SUBAPPLICATION Uebung_237_AX (* AD_TO_AR-Bitfalle: derselbe Analogwert einmal FALSCH ueber AD_TO_AR (Bit-Reinterpretation) und einmal RICHTIG ueber AD_TO_AR_NUM (echter numerischer Cast) gelesen *)
  (* Standard: 61499-2; Description: Copyright (c) 2026 Meisterschulen am Ostbahnhof This program and the accompanying materials are made available under the terms of the Eclipse Public License 2.0 which is available at https://www.eclipse.org/legal/epl-2.0/ SPDX-License-Identifier: EPL-2.0 *)
  (* Version 1.0, 2026-09-07, Franz Höpfinger, Meisterschulen am Ostbahnhof, initial API and implementation and/or initial documentation *)
  PACKAGE Uebungen;
  IMPORT logiBUS::io::AI::logiBUS_AI::AnalogInput_I4;
  (* Documentation:
  AD_TO_AR-Bitfalle: Bit-Reinterpretation vs. numerischer Cast
   Derselbe rohe Analogwert (AnalogInput_I4, ueber AD_SPLIT_2 verdoppelt) wird hier auf zwei Arten von AD (DWORD-Adapter) nach AR (REAL-Adapter) konvertiert:
    - AD_TO_AR_WRONG (AD_TO_AR): sieht wie die naheliegende direkte Konvertierung aus, ist intern aber F_DWORD_TO_REAL - eine reine IEEE754-Bit-Reinterpretation. Ein roher Analogwert wie DWORD#2048 wird dadurch NICHT zu REAL#2048.0, sondern zu einer bedeutungslosen Zahl nahe Null.
   - AD_TO_AR_NUM_CORRECT (AD_TO_AR_NUM): macht denselben Job numerisch korrekt, ueber die Zwischenkette DWORD->UDINT->REAL (dieselbe Kette, die Uebung_028a_AR von Hand aus AD_TO_AUDI+AUDI_TO_AR zusammensetzt - AD_TO_AR_NUM ist das drop-in-kompatible Einzelbaustein-Aequivalent).
    Arbeitsauftrag
   Beide AR_OUT.D1-Pins im laufenden 4diac-Monitor beobachten (rechte Maustaste auf den Pin -> Watch) und vergleichen: AD_TO_AR_WRONG zeigt eine kleine, mit dem tatsaechlichen Analogwert scheinbar unzusammenhaengende Zahl; AD_TO_AR_NUM_CORRECT zeigt den plausiblen, tatsaechlichen Messwert. Erklaeren Sie, warum der "direkt aussehende" Weg (AD_TO_AR) hier der falsche ist - siehe auch die Dokumentation in AD_TO_AR.fbt selbst, die genau vor dieser Falle warnt.
   Wann ist AD_TO_AR trotzdem richtig?
   Wenn AD_IN bereits ein Bitmuster ist, das als REAL gemeint war (z.B. das Ergebnis von F_REAL_TO_DWORD an anderer Stelle) - dann ist die Bit-Reinterpretation genau die richtige, verlustfreie Rueckrichtung. Ein roher Analog-/Zaehlerwert wie in dieser Uebung ist das Gegenbeispiel: hier ist der numerische Cast (AD_TO_AR_NUM) richtig.
  *)
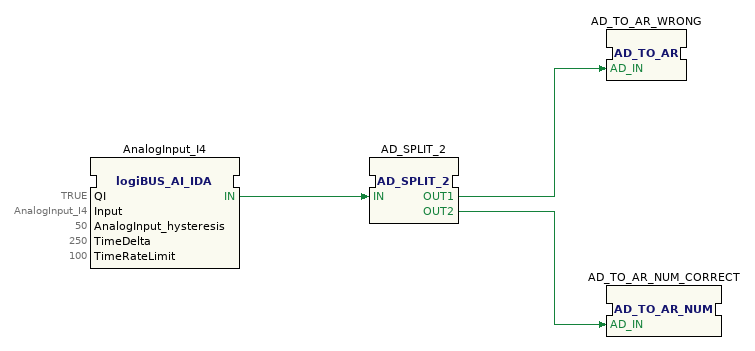
  (* FALSCH: AD_TO_AR ist eine reine IEEE754-Bit-Reinterpretation (F_DWORD_TO_REAL), kein numerischer Cast. Derselbe Analog-Rohwert, der ueber AD_TO_AR_NUM_CORRECT (unten) den richtigen Zahlenwert liefert, ergibt hier eine bedeutungslose Zahl nahe Null. AR_OUT.D1 beider Bausteine im 4diac-Monitor beobachten (rechte Maustaste auf den Pin -> Watch) und vergleichen. *)
  FBS
    AnalogInput_I4 : logiBUS::io::AI::logiBUS_AI_IDA(QI := TRUE, Input := AnalogInput_I4, AnalogInput_hysteresis := 50, TimeDelta := 250, TimeRateLimit := 100);
    AD_SPLIT_2 : adapter::events::unidirectional::AD_SPLIT_2;
    AD_TO_AR_WRONG : adapter::conversion::unidirectional::AD_TO_AR;
    AD_TO_AR_NUM_CORRECT : adapter::conversion::unidirectional::AD_TO_AR_NUM;
  END_FBS
  ADAPTER_CONNECTIONS
    AnalogInput_I4.IN TO AD_SPLIT_2.IN;
    AD_SPLIT_2.OUT1 TO AD_TO_AR_WRONG.AD_IN;
    AD_SPLIT_2.OUT2 TO AD_TO_AR_NUM_CORRECT.AD_IN;
  END_CONNECTIONS
END_SUBAPPLICATION
